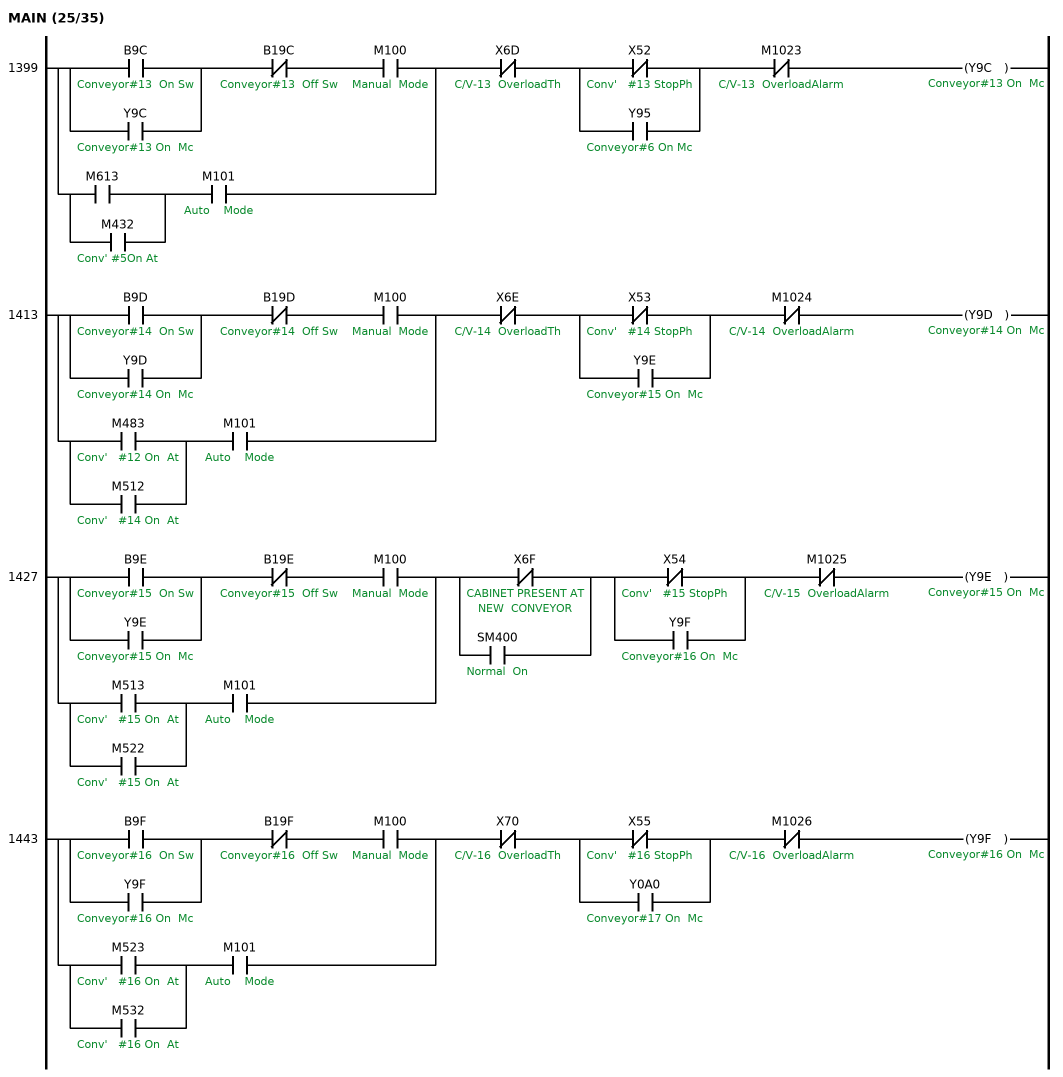
[picture p24: ladder of MAIN, rungs at steps 1399 to 1443]
1399  LD      B9C  ; Conveyor#13  On Sw
      OR      Y9C  ; Conveyor#13 On  Mc
      ANI     B19C  ; Conveyor#13  Off Sw
      AND     M100  ; Manual  Mode
      LD      M613
      OR      M432  ; Conv' #5On At
      AND     M101  ; Auto    Mode
      ORB
      ANI     X6D  ; C/V-13  OverloadTh
      LDI     X52  ; Conv'   #13 StopPh
      OR      Y95  ; Conveyor#6 On Mc
      ANB
      ANI     M1023  ; C/V-13  OverloadAlarm
      OUT     Y9C  ; Conveyor#13 On  Mc
1413  LD      B9D  ; Conveyor#14  On Sw
      OR      Y9D  ; Conveyor#14 On  Mc
      ANI     B19D  ; Conveyor#14  Off Sw
      AND     M100  ; Manual  Mode
      LD      M483  ; Conv'   #12 On  At
      OR      M512  ; Conv'   #14 On  At
      AND     M101  ; Auto    Mode
      ORB
      ANI     X6E  ; C/V-14  OverloadTh
      LDI     X53  ; Conv'   #14 StopPh
      OR      Y9E  ; Conveyor#15 On  Mc
      ANB
      ANI     M1024  ; C/V-14  OverloadAlarm
      OUT     Y9D  ; Conveyor#14 On  Mc
1427  LD      B9E  ; Conveyor#15  On Sw
      OR      Y9E  ; Conveyor#15 On  Mc
      ANI     B19E  ; Conveyor#15  Off Sw
      AND     M100  ; Manual  Mode
      LD      M513  ; Conv'   #15 On  At
      OR      M522  ; Conv'   #15 On  At
      AND     M101  ; Auto    Mode
      ORB
      LDI     X6F  ; CABINET PRESENT AT NEW  CONVEYOR
      OR      SM400  ; Normal  On
      ANB
      LDI     X54  ; Conv'   #15 StopPh
      OR      Y9F  ; Conveyor#16 On  Mc
      ANB
      ANI     M1025  ; C/V-15  OverloadAlarm
      OUT     Y9E  ; Conveyor#15 On  Mc
1443  LD      B9F  ; Conveyor#16  On Sw
      OR      Y9F  ; Conveyor#16 On  Mc
      ANI     B19F  ; Conveyor#16  Off Sw
      AND     M100  ; Manual  Mode
      LD      M523  ; Conv'   #16 On  At
      OR      M532  ; Conv'   #16 On  At
      AND     M101  ; Auto    Mode
      ORB
      ANI     X70  ; C/V-16  OverloadTh
      LDI     X55  ; Conv'   #16 StopPh
      OR      Y0A0  ; Conveyor#17 On  Mc
      ANB
      ANI     M1026  ; C/V-16  OverloadAlarm
      OUT     Y9F  ; Conveyor#16 On  Mc
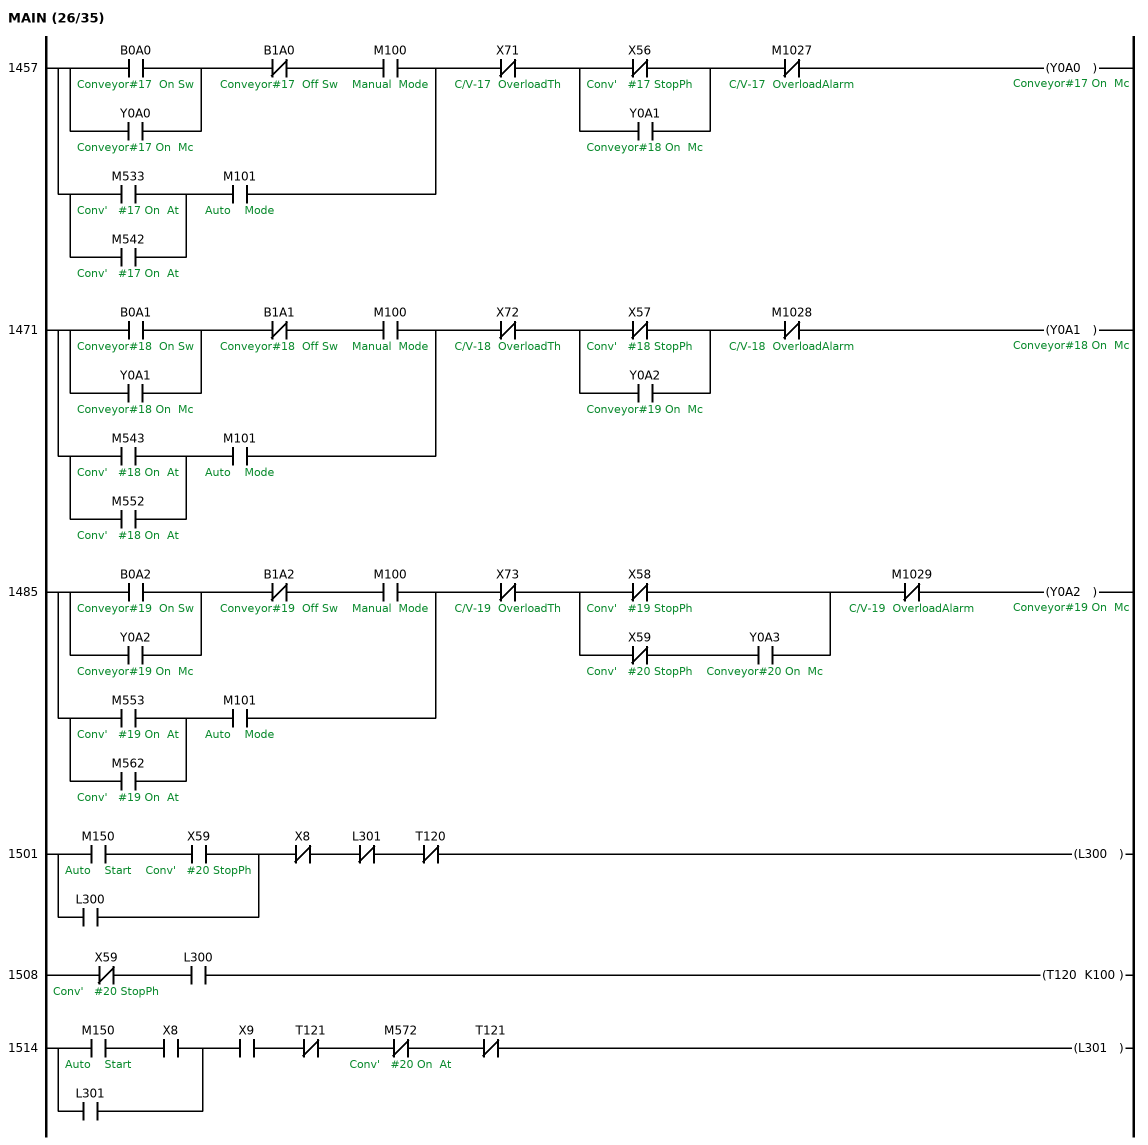
1457  LD      B0A0  ; Conveyor#17  On Sw
      OR      Y0A0  ; Conveyor#17 On  Mc
      ANI     B1A0  ; Conveyor#17  Off Sw
      AND     M100  ; Manual  Mode
      LD      M533  ; Conv'   #17 On  At
      OR      M542  ; Conv'   #17 On  At
      AND     M101  ; Auto    Mode
      ORB
      ANI     X71  ; C/V-17  OverloadTh
      LDI     X56  ; Conv'   #17 StopPh
      OR      Y0A1  ; Conveyor#18 On  Mc
      ANB
      ANI     M1027  ; C/V-17  OverloadAlarm
      OUT     Y0A0  ; Conveyor#17 On  Mc
1471  LD      B0A1  ; Conveyor#18  On Sw
      OR      Y0A1  ; Conveyor#18 On  Mc
      ANI     B1A1  ; Conveyor#18  Off Sw
      AND     M100  ; Manual  Mode
      LD      M543  ; Conv'   #18 On  At
      OR      M552  ; Conv'   #18 On  At
      AND     M101  ; Auto    Mode
      ORB
      ANI     X72  ; C/V-18  OverloadTh
      LDI     X57  ; Conv'   #18 StopPh
      OR      Y0A2  ; Conveyor#19 On  Mc
      ANB
      ANI     M1028  ; C/V-18  OverloadAlarm
      OUT     Y0A1  ; Conveyor#18 On  Mc
1485  LD      B0A2  ; Conveyor#19  On Sw
      OR      Y0A2  ; Conveyor#19 On  Mc
      ANI     B1A2  ; Conveyor#19  Off Sw
      AND     M100  ; Manual  Mode
      LD      M553  ; Conv'   #19 On  At
      OR      M562  ; Conv'   #19 On  At
      AND     M101  ; Auto    Mode
      ORB
      ANI     X73  ; C/V-19  OverloadTh
      LDI     X58  ; Conv'   #19 StopPh
      LDI     X59  ; Conv'   #20 StopPh
      AND     Y0A3  ; Conveyor#20 On  Mc
      ORB
      ANB
      ANI     M1029  ; C/V-19  OverloadAlarm
      OUT     Y0A2  ; Conveyor#19 On  Mc
1501  LD      M150  ; Auto    Start
      AND     X59  ; Conv'   #20 StopPh
      OR      L300
      ANI     X8
      ANI     L301
      ANI     T120
      OUT     L300
1508  LDI     X59  ; Conv'   #20 StopPh
      AND     L300
      OUT     T120 K100
1514  LD      M150  ; Auto    Start
      AND     X8
      OR      L301
      AND     X9
      ANI     T121
      ANI     M572  ; Conv'   #20 On  At
      ANI     T121
      OUT     L301
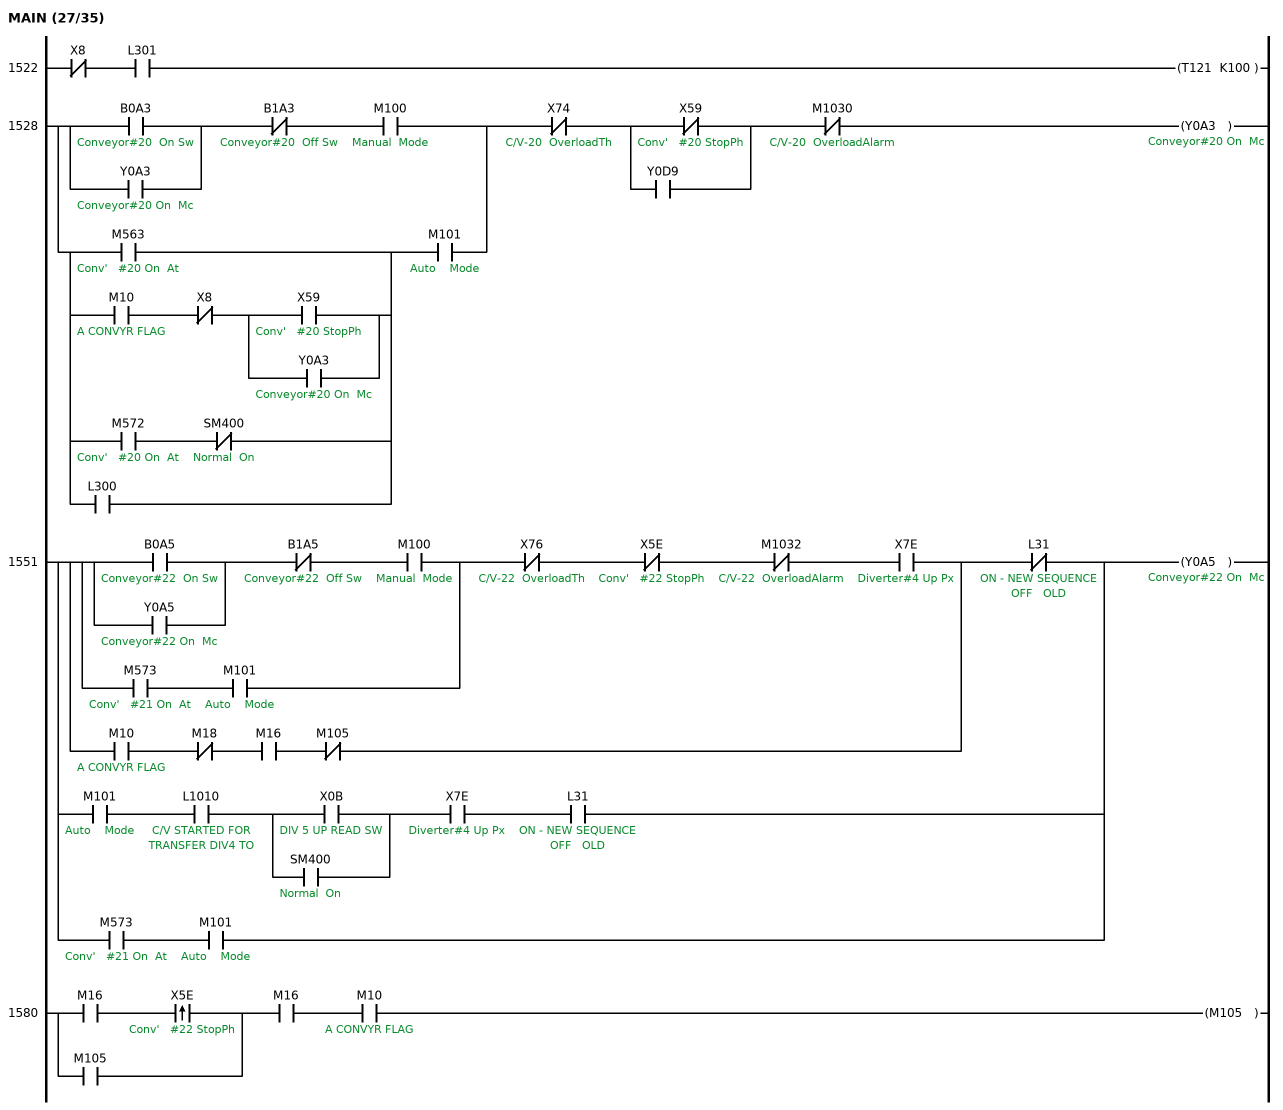
1522  LDI     X8
      AND     L301
      OUT     T121 K100
1528  LD      B0A3  ; Conveyor#20  On Sw
      OR      Y0A3  ; Conveyor#20 On  Mc
      ANI     B1A3  ; Conveyor#20  Off Sw
      AND     M100  ; Manual  Mode
      LD      M563  ; Conv'   #20 On  At
      LD      M10  ; A CONVYR FLAG
      ANI     X8
      LD      X59  ; Conv'   #20 StopPh
      OR      Y0A3  ; Conveyor#20 On  Mc
      ANB
      ORB
      LD      M572  ; Conv'   #20 On  At
      ANI     SM400  ; Normal  On
      ORB
      OR      L300
      AND     M101  ; Auto    Mode
      ORB
      ANI     X74  ; C/V-20  OverloadTh
      LDI     X59  ; Conv'   #20 StopPh
      OR      Y0D9
      ANB
      ANI     M1030  ; C/V-20  OverloadAlarm
      OUT     Y0A3  ; Conveyor#20 On  Mc
1551  LD      B0A5  ; Conveyor#22  On Sw
      OR      Y0A5  ; Conveyor#22 On  Mc
      ANI     B1A5  ; Conveyor#22  Off Sw
      AND     M100  ; Manual  Mode
      LD      M573  ; Conv'   #21 On  At
      AND     M101  ; Auto    Mode
      ORB
      ANI     X76  ; C/V-22  OverloadTh
      ANI     X5E  ; Conv'   #22 StopPh
      ANI     M1032  ; C/V-22  OverloadAlarm
      AND     X7E  ; Diverter#4 Up Px
      LD      M10  ; A CONVYR FLAG
      ANI     M18
      AND     M16
      ANI     M105
      ORB
      ANI     L31  ; ON - NEW SEQUENCE OFF   OLD
      LD      M101  ; Auto    Mode
      AND     L1010  ; C/V STARTED FOR TRANSFER DIV4 TO
      LD      X0B  ; DIV 5 UP READ SW
      OR      SM400  ; Normal  On
      ANB
      AND     X7E  ; Diverter#4 Up Px
      AND     L31  ; ON - NEW SEQUENCE OFF   OLD
      ORB
      LD      M573  ; Conv'   #21 On  At
      AND     M101  ; Auto    Mode
      ORB
      OUT     Y0A5  ; Conveyor#22 On  Mc
1580  LD      M16
      ANDP    X5E  ; Conv'   #22 StopPh
      OR      M105
      AND     M16
      AND     M10  ; A CONVYR FLAG
      OUT     M105
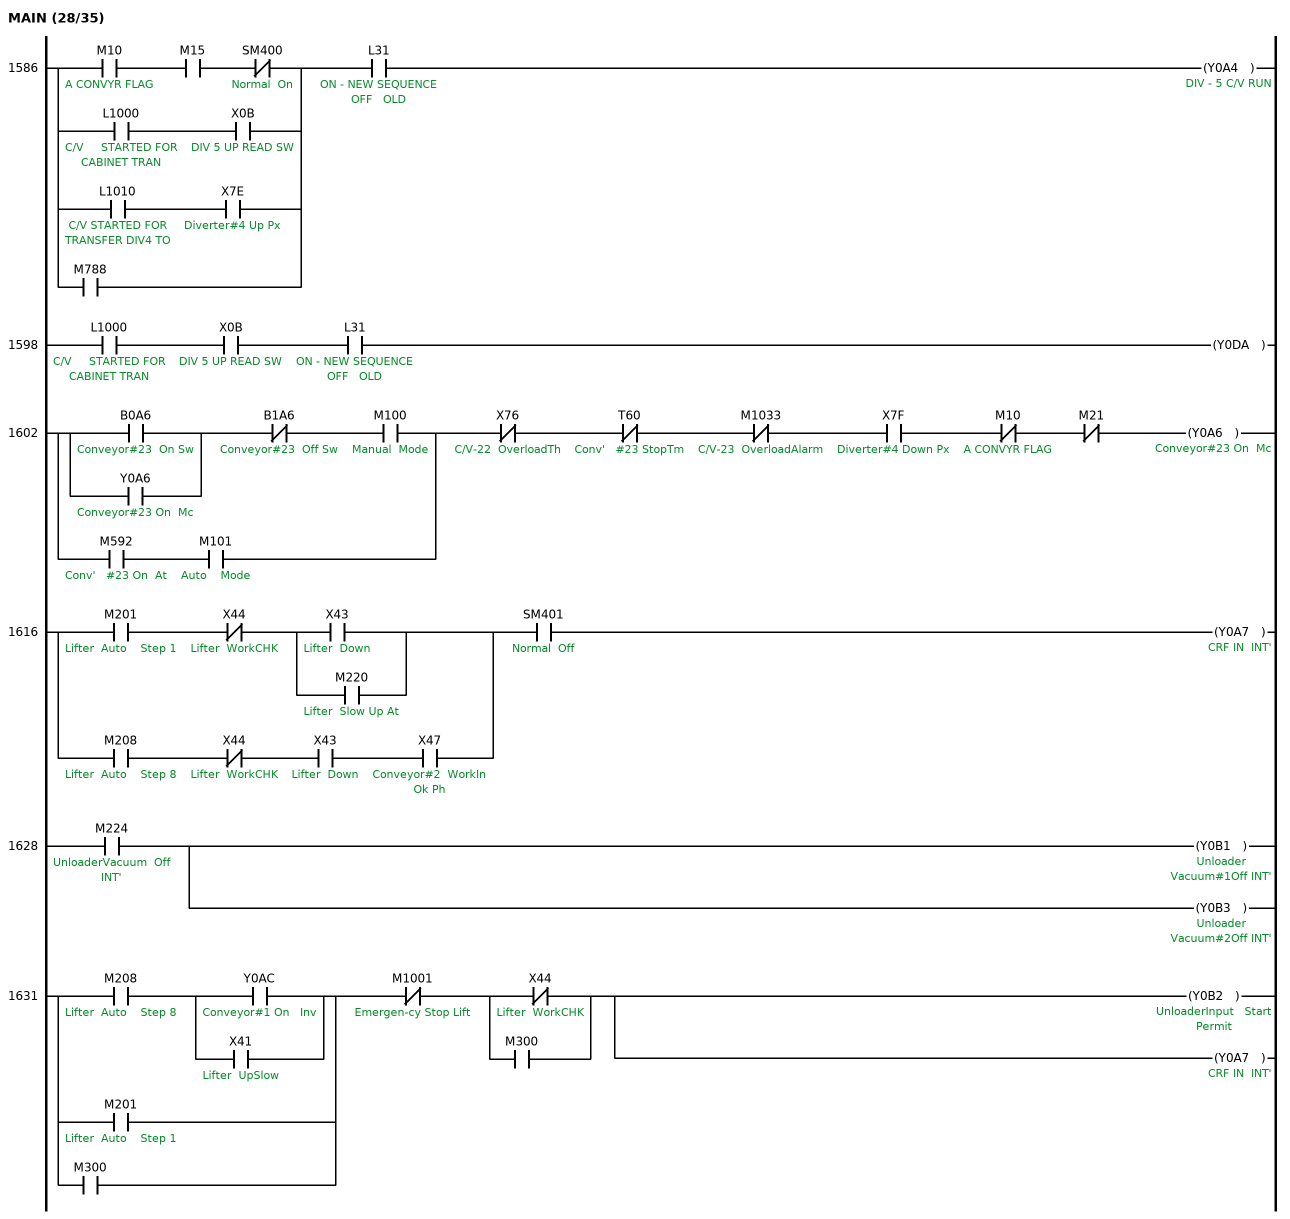
1586  LD      M10  ; A CONVYR FLAG
      AND     M15
      ANI     SM400  ; Normal  On
      LD      L1000  ; C/V     STARTED FOR CABINET TRAN
      AND     X0B  ; DIV 5 UP READ SW
      ORB
      LD      L1010  ; C/V STARTED FOR TRANSFER DIV4 TO
      AND     X7E  ; Diverter#4 Up Px
      ORB
      OR      M788
      AND     L31  ; ON - NEW SEQUENCE OFF   OLD
      OUT     Y0A4  ; DIV - 5 C/V RUN
1598  LD      L1000  ; C/V     STARTED FOR CABINET TRAN
      AND     X0B  ; DIV 5 UP READ SW
      AND     L31  ; ON - NEW SEQUENCE OFF   OLD
      OUT     Y0DA
1602  LD      B0A6  ; Conveyor#23  On Sw
      OR      Y0A6  ; Conveyor#23 On  Mc
      ANI     B1A6  ; Conveyor#23  Off Sw
      AND     M100  ; Manual  Mode
      LD      M592  ; Conv'   #23 On  At
      AND     M101  ; Auto    Mode
      ORB
      ANI     X76  ; C/V-22  OverloadTh
      ANI     T60  ; Conv'   #23 StopTm
      ANI     M1033  ; C/V-23  OverloadAlarm
      AND     X7F  ; Diverter#4 Down Px
      ANI     M10  ; A CONVYR FLAG
      ANI     M21
      OUT     Y0A6  ; Conveyor#23 On  Mc
1616  LD      M201  ; Lifter  Auto    Step 1
      ANI     X44  ; Lifter  WorkCHK
      LD      X43  ; Lifter  Down
      OR      M220  ; Lifter  Slow Up At
      ANB
      LD      M208  ; Lifter  Auto    Step 8
      ANI     X44  ; Lifter  WorkCHK
      AND     X43  ; Lifter  Down
      AND     X47  ; Conveyor#2  WorkIn Ok Ph
      ORB
      AND     SM401  ; Normal  Off
      OUT     Y0A7  ; CRF IN  INT'
1628  LD      M224  ; UnloaderVacuum  Off INT'
      OUT     Y0B1  ; UnloaderVacuum#1Off INT'
      OUT     Y0B3  ; UnloaderVacuum#2Off INT'
1631  LD      M208  ; Lifter  Auto    Step 8
      LD      Y0AC  ; Conveyor#1 On   Inv
      OR      X41  ; Lifter  UpSlow
      ANB
      OR      M201  ; Lifter  Auto    Step 1
      OR      M300
      ANI     M1001  ; Emergen-cy Stop Lift
      LDI     X44  ; Lifter  WorkCHK
      OR      M300
      ANB
      OUT     Y0B2  ; UnloaderInput   Start   Permit
      OUT     Y0A7  ; CRF IN  INT'
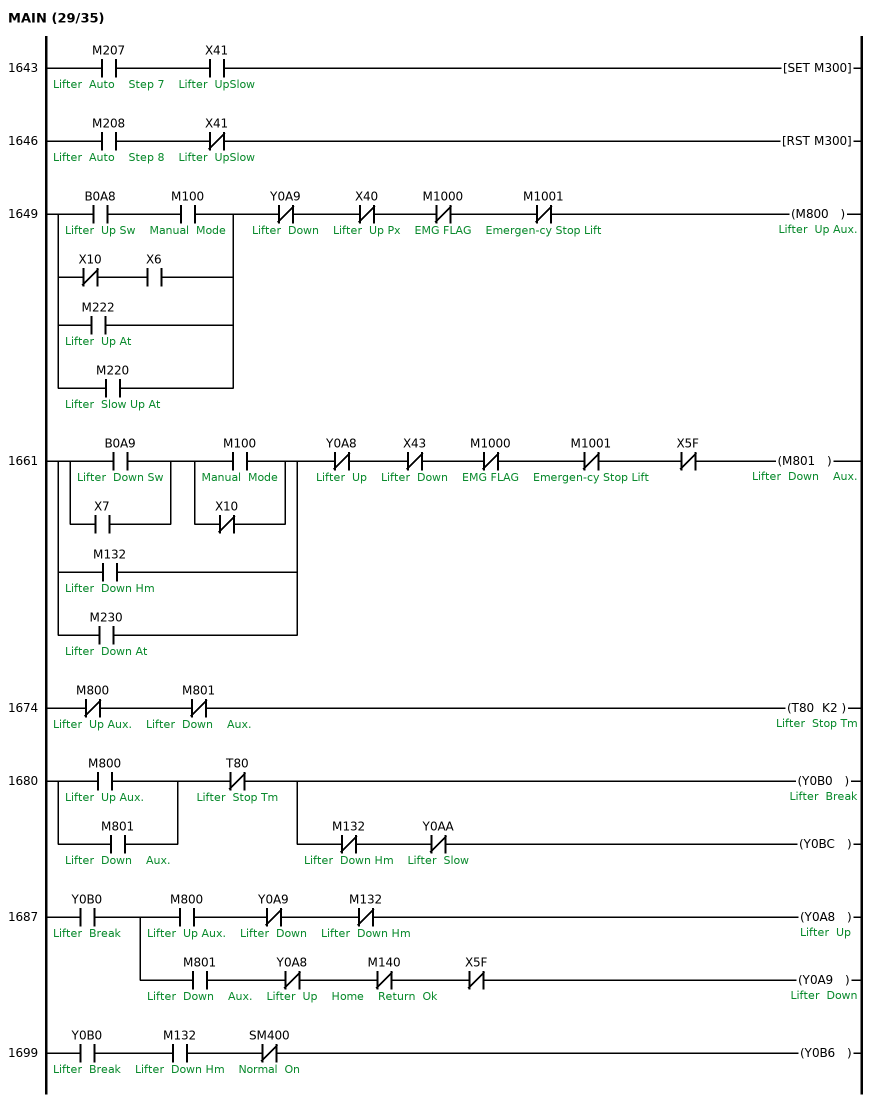
1643  LD      M207  ; Lifter  Auto    Step 7
      AND     X41  ; Lifter  UpSlow
      SET     M300
1646  LD      M208  ; Lifter  Auto    Step 8
      ANI     X41  ; Lifter  UpSlow
      RST     M300
1649  LD      B0A8  ; Lifter  Up Sw
      AND     M100  ; Manual  Mode
      LDI     X10
      AND     X6
      ORB
      OR      M222  ; Lifter  Up At
      OR      M220  ; Lifter  Slow Up At
      ANI     Y0A9  ; Lifter  Down
      ANI     X40  ; Lifter  Up Px
      ANI     M1000  ; EMG FLAG
      ANI     M1001  ; Emergen-cy Stop Lift
      OUT     M800  ; Lifter  Up Aux.
1661  LD      B0A9  ; Lifter  Down Sw
      OR      X7
      LD      M100  ; Manual  Mode
      ORI     X10
      ANB
      OR      M132  ; Lifter  Down Hm
      OR      M230  ; Lifter  Down At
      ANI     Y0A8  ; Lifter  Up
      ANI     X43  ; Lifter  Down
      ANI     M1000  ; EMG FLAG
      ANI     M1001  ; Emergen-cy Stop Lift
      ANI     X5F
      OUT     M801  ; Lifter  Down    Aux.
1674  LDI     M800  ; Lifter  Up Aux.
      ANI     M801  ; Lifter  Down    Aux.
      OUT     T80 K2  ; Lifter  Stop Tm
1680  LD      M800  ; Lifter  Up Aux.
      OR      M801  ; Lifter  Down    Aux.
      ANI     T80  ; Lifter  Stop Tm
      OUT     Y0B0  ; Lifter  Break
      ANI     M132  ; Lifter  Down Hm
      ANI     Y0AA  ; Lifter  Slow
      OUT     Y0BC
1687  LD      Y0B0  ; Lifter  Break
      MPS
      AND     M800  ; Lifter  Up Aux.
      ANI     Y0A9  ; Lifter  Down
      ANI     M132  ; Lifter  Down Hm
      OUT     Y0A8  ; Lifter  Up
      MPP
      AND     M801  ; Lifter  Down    Aux.
      ANI     Y0A8  ; Lifter  Up
      ANI     M140  ; Home    Return  Ok
      ANI     X5F
      OUT     Y0A9  ; Lifter  Down
1699  LD      Y0B0  ; Lifter  Break
      AND     M132  ; Lifter  Down Hm
      ANI     SM400  ; Normal  On
      OUT     Y0B6
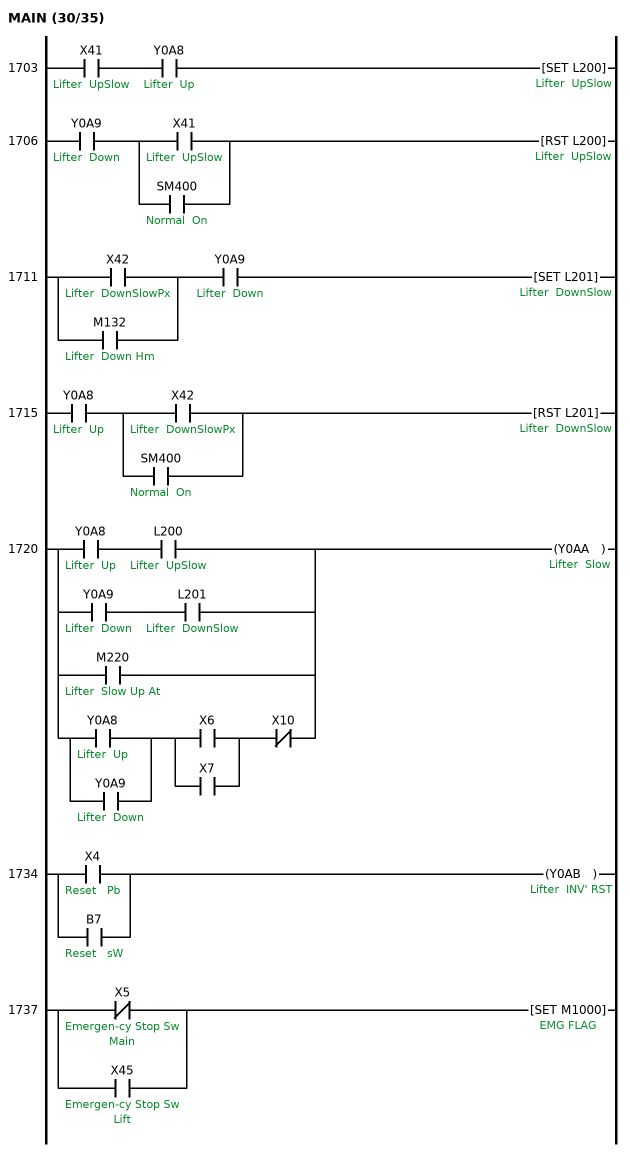
1703  LD      X41  ; Lifter  UpSlow
      AND     Y0A8  ; Lifter  Up
      SET     L200  ; Lifter  UpSlow
1706  LD      Y0A9  ; Lifter  Down
      LD      X41  ; Lifter  UpSlow
      OR      SM400  ; Normal  On
      ANB
      RST     L200  ; Lifter  UpSlow
1711  LD      X42  ; Lifter  DownSlowPx
      OR      M132  ; Lifter  Down Hm
      AND     Y0A9  ; Lifter  Down
      SET     L201  ; Lifter  DownSlow
1715  LD      Y0A8  ; Lifter  Up
      LD      X42  ; Lifter  DownSlowPx
      OR      SM400  ; Normal  On
      ANB
      RST     L201  ; Lifter  DownSlow
1720  LD      Y0A8  ; Lifter  Up
      AND     L200  ; Lifter  UpSlow
      LD      Y0A9  ; Lifter  Down
      AND     L201  ; Lifter  DownSlow
      ORB
      OR      M220  ; Lifter  Slow Up At
      LD      Y0A8  ; Lifter  Up
      OR      Y0A9  ; Lifter  Down
      LD      X6
      OR      X7
      ANB
      ANI     X10
      ORB
      OUT     Y0AA  ; Lifter  Slow
1734  LD      X4  ; Reset   Pb
      OR      B7  ; Reset   sW
      OUT     Y0AB  ; Lifter  INV' RST
1737  LDI     X5  ; Emergen-cy Stop Sw Main
      OR      X45  ; Emergen-cy Stop Sw Lift
      SET     M1000  ; EMG FLAG
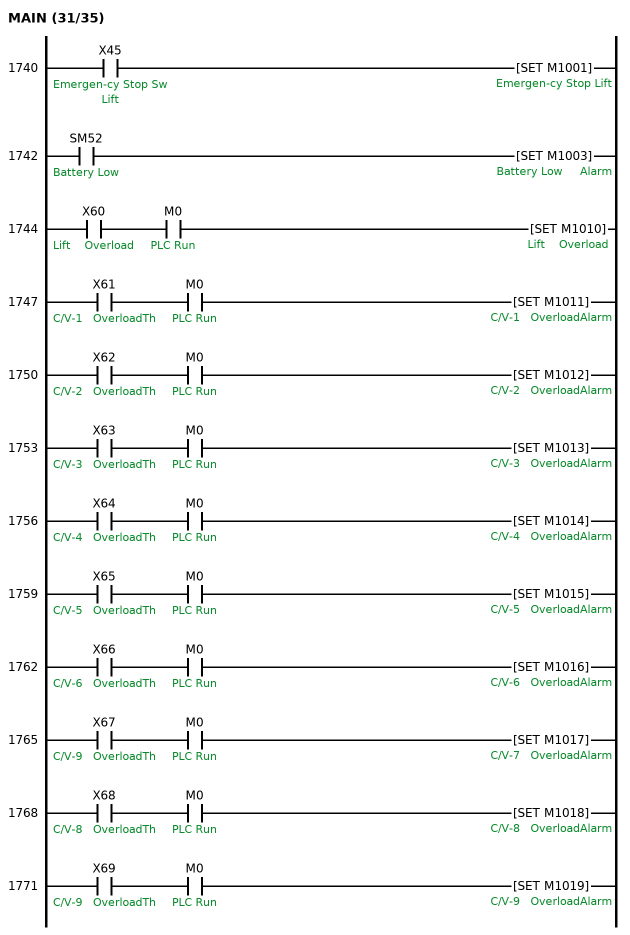
1740  LD      X45  ; Emergen-cy Stop Sw Lift
      SET     M1001  ; Emergen-cy Stop Lift
1742  LD      SM52  ; Battery Low
      SET     M1003  ; Battery Low     Alarm
1744  LD      X60  ; Lift    Overload
      AND     M0  ; PLC Run
      SET     M1010  ; Lift    Overload
1747  LD      X61  ; C/V-1   OverloadTh
      AND     M0  ; PLC Run
      SET     M1011  ; C/V-1   OverloadAlarm
1750  LD      X62  ; C/V-2   OverloadTh
      AND     M0  ; PLC Run
      SET     M1012  ; C/V-2   OverloadAlarm
1753  LD      X63  ; C/V-3   OverloadTh
      AND     M0  ; PLC Run
      SET     M1013  ; C/V-3   OverloadAlarm
1756  LD      X64  ; C/V-4   OverloadTh
      AND     M0  ; PLC Run
      SET     M1014  ; C/V-4   OverloadAlarm
1759  LD      X65  ; C/V-5   OverloadTh
      AND     M0  ; PLC Run
      SET     M1015  ; C/V-5   OverloadAlarm
1762  LD      X66  ; C/V-6   OverloadTh
      AND     M0  ; PLC Run
      SET     M1016  ; C/V-6   OverloadAlarm
1765  LD      X67  ; C/V-9   OverloadTh
      AND     M0  ; PLC Run
      SET     M1017  ; C/V-7   OverloadAlarm
1768  LD      X68  ; C/V-8   OverloadTh
      AND     M0  ; PLC Run
      SET     M1018  ; C/V-8   OverloadAlarm
1771  LD      X69  ; C/V-9   OverloadTh
      AND     M0  ; PLC Run
      SET     M1019  ; C/V-9   OverloadAlarm
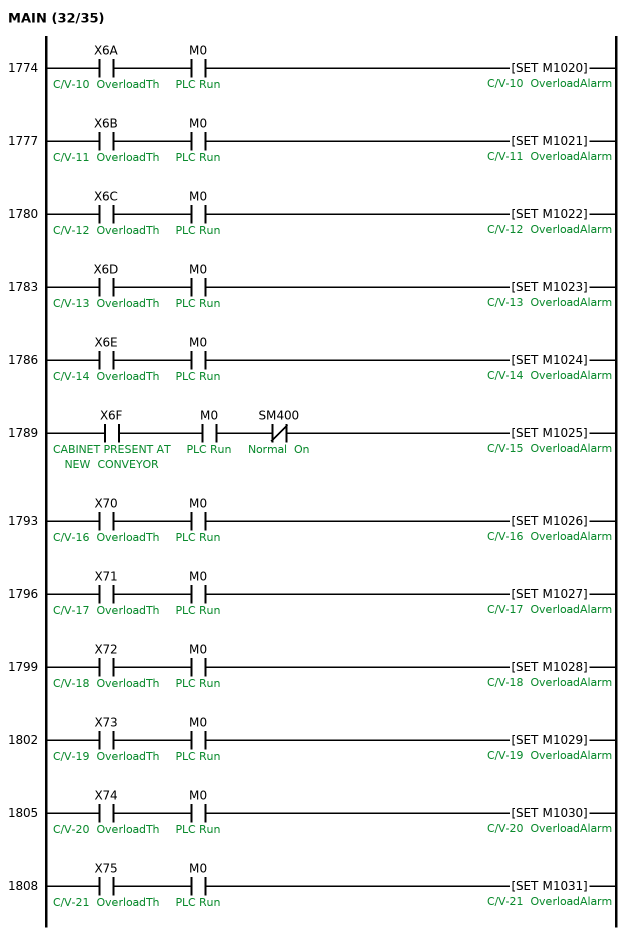
1774  LD      X6A  ; C/V-10  OverloadTh
      AND     M0  ; PLC Run
      SET     M1020  ; C/V-10  OverloadAlarm
1777  LD      X6B  ; C/V-11  OverloadTh
      AND     M0  ; PLC Run
      SET     M1021  ; C/V-11  OverloadAlarm
1780  LD      X6C  ; C/V-12  OverloadTh
      AND     M0  ; PLC Run
      SET     M1022  ; C/V-12  OverloadAlarm
1783  LD      X6D  ; C/V-13  OverloadTh
      AND     M0  ; PLC Run
      SET     M1023  ; C/V-13  OverloadAlarm
1786  LD      X6E  ; C/V-14  OverloadTh
      AND     M0  ; PLC Run
      SET     M1024  ; C/V-14  OverloadAlarm
1789  LD      X6F  ; CABINET PRESENT AT NEW  CONVEYOR
      AND     M0  ; PLC Run
      ANI     SM400  ; Normal  On
      SET     M1025  ; C/V-15  OverloadAlarm
1793  LD      X70  ; C/V-16  OverloadTh
      AND     M0  ; PLC Run
      SET     M1026  ; C/V-16  OverloadAlarm
1796  LD      X71  ; C/V-17  OverloadTh
      AND     M0  ; PLC Run
      SET     M1027  ; C/V-17  OverloadAlarm
1799  LD      X72  ; C/V-18  OverloadTh
      AND     M0  ; PLC Run
      SET     M1028  ; C/V-18  OverloadAlarm
1802  LD      X73  ; C/V-19  OverloadTh
      AND     M0  ; PLC Run
      SET     M1029  ; C/V-19  OverloadAlarm
1805  LD      X74  ; C/V-20  OverloadTh
      AND     M0  ; PLC Run
      SET     M1030  ; C/V-20  OverloadAlarm
1808  LD      X75  ; C/V-21  OverloadTh
      AND     M0  ; PLC Run
      SET     M1031  ; C/V-21  OverloadAlarm
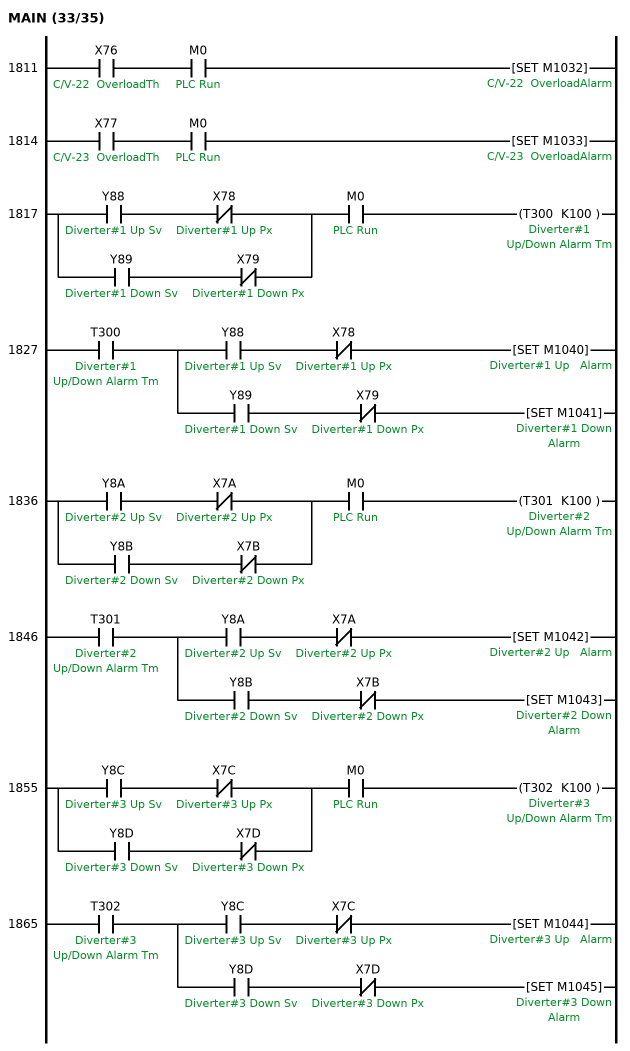
1811  LD      X76  ; C/V-22  OverloadTh
      AND     M0  ; PLC Run
      SET     M1032  ; C/V-22  OverloadAlarm
1814  LD      X77  ; C/V-23  OverloadTh
      AND     M0  ; PLC Run
      SET     M1033  ; C/V-23  OverloadAlarm
1817  LD      Y88  ; Diverter#1 Up Sv
      ANI     X78  ; Diverter#1 Up Px
      LD      Y89  ; Diverter#1 Down Sv
      ANI     X79  ; Diverter#1 Down Px
      ORB
      AND     M0  ; PLC Run
      OUT     T300 K100  ; Diverter#1      Up/Down Alarm Tm
1827  LD      T300  ; Diverter#1      Up/Down Alarm Tm
      MPS
      AND     Y88  ; Diverter#1 Up Sv
      ANI     X78  ; Diverter#1 Up Px
      SET     M1040  ; Diverter#1 Up   Alarm
      MPP
      AND     Y89  ; Diverter#1 Down Sv
      ANI     X79  ; Diverter#1 Down Px
      SET     M1041  ; Diverter#1 Down Alarm
1836  LD      Y8A  ; Diverter#2 Up Sv
      ANI     X7A  ; Diverter#2 Up Px
      LD      Y8B  ; Diverter#2 Down Sv
      ANI     X7B  ; Diverter#2 Down Px
      ORB
      AND     M0  ; PLC Run
      OUT     T301 K100  ; Diverter#2      Up/Down Alarm Tm
1846  LD      T301  ; Diverter#2      Up/Down Alarm Tm
      MPS
      AND     Y8A  ; Diverter#2 Up Sv
      ANI     X7A  ; Diverter#2 Up Px
      SET     M1042  ; Diverter#2 Up   Alarm
      MPP
      AND     Y8B  ; Diverter#2 Down Sv
      ANI     X7B  ; Diverter#2 Down Px
      SET     M1043  ; Diverter#2 Down Alarm
1855  LD      Y8C  ; Diverter#3 Up Sv
      ANI     X7C  ; Diverter#3 Up Px
      LD      Y8D  ; Diverter#3 Down Sv
      ANI     X7D  ; Diverter#3 Down Px
      ORB
      AND     M0  ; PLC Run
      OUT     T302 K100  ; Diverter#3      Up/Down Alarm Tm
1865  LD      T302  ; Diverter#3      Up/Down Alarm Tm
      MPS
      AND     Y8C  ; Diverter#3 Up Sv
      ANI     X7C  ; Diverter#3 Up Px
      SET     M1044  ; Diverter#3 Up   Alarm
      MPP
      AND     Y8D  ; Diverter#3 Down Sv
      ANI     X7D  ; Diverter#3 Down Px
      SET     M1045  ; Diverter#3 Down Alarm
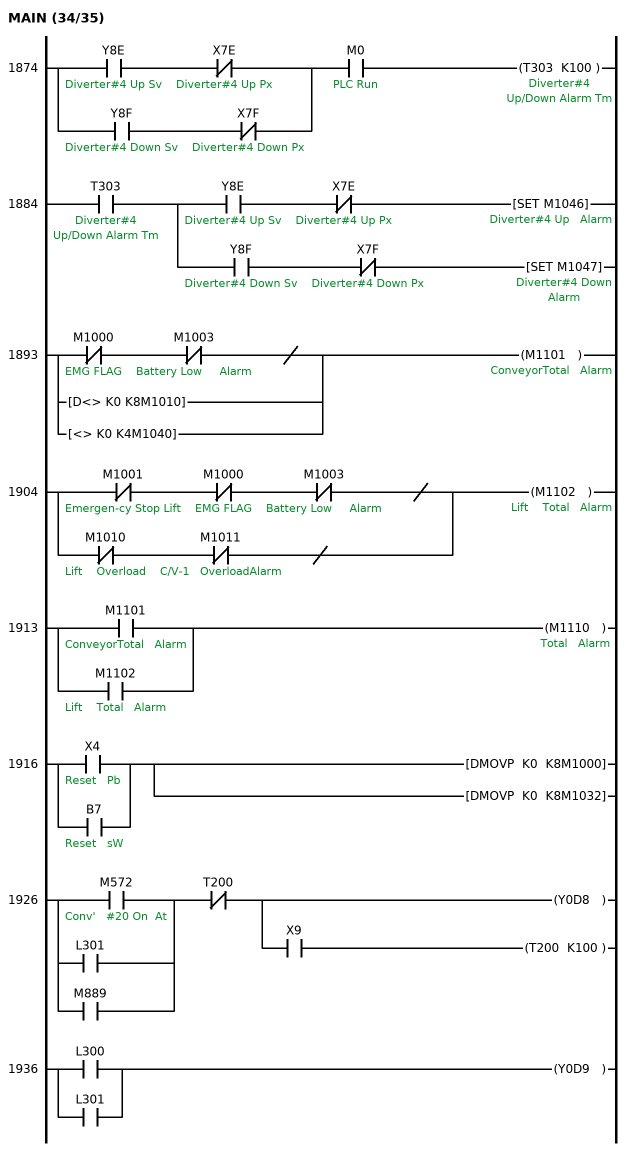
1874  LD      Y8E  ; Diverter#4 Up Sv
      ANI     X7E  ; Diverter#4 Up Px
      LD      Y8F  ; Diverter#4 Down Sv
      ANI     X7F  ; Diverter#4 Down Px
      ORB
      AND     M0  ; PLC Run
      OUT     T303 K100  ; Diverter#4      Up/Down Alarm Tm
1884  LD      T303  ; Diverter#4      Up/Down Alarm Tm
      MPS
      AND     Y8E  ; Diverter#4 Up Sv
      ANI     X7E  ; Diverter#4 Up Px
      SET     M1046  ; Diverter#4 Up   Alarm
      MPP
      AND     Y8F  ; Diverter#4 Down Sv
      ANI     X7F  ; Diverter#4 Down Px
      SET     M1047  ; Diverter#4 Down Alarm
1893  LDI     M1000  ; EMG FLAG
      ANI     M1003  ; Battery Low     Alarm
      INV
      ORD<>   K0 K8M1010  ; Lift    Overload
      OR<>    K0 K4M1040  ; Diverter#1 Up   Alarm
      OUT     M1101  ; ConveyorTotal   Alarm
1904  LDI     M1001  ; Emergen-cy Stop Lift
      ANI     M1000  ; EMG FLAG
      ANI     M1003  ; Battery Low     Alarm
      INV
      LDI     M1010  ; Lift    Overload
      ANI     M1011  ; C/V-1   OverloadAlarm
      INV
      ORB
      OUT     M1102  ; Lift    Total   Alarm
1913  LD      M1101  ; ConveyorTotal   Alarm
      OR      M1102  ; Lift    Total   Alarm
      OUT     M1110  ; Total   Alarm
1916  LD      X4  ; Reset   Pb
      OR      B7  ; Reset   sW
      DMOVP   K0 K8M1000
      DMOVP   K0 K8M1032
1926  LD      M572  ; Conv'   #20 On  At
      OR      L301
      OR      M889
      ANI     T200
      OUT     Y0D8
      AND     X9
      OUT     T200 K100
1936  LD      L300
      OR      L301
      OUT     Y0D9
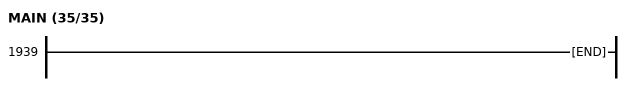
1939  END
END_PROGRAM

// device comments not shown above
Y0BA  ; TRANSER C/V     RUNNING
Y0BB  ; DIVERTOR C/V    RUNNING
Y732  ; PANEL ATB SIDE
M582  ; Conv'   #21 On  At
M583  ; Conv'   #22 On  At
B0A4  ; Conveyor#21  On Sw
B1A4  ; Conveyor#21  OffSw
